(* IEC 61131-3 sources: inproshop/test13_exported/1.Function/FC, 5 files *)

(* ---- FC_AryCmp.st ---- *)
FUNCTION FC_AryCmp : BOOL
VAR_INPUT
	iAry1:ARRAY[0..50]OF BOOL;
	iAry2:ARRAY[0..50]OF BOOL;
END_VAR
VAR
	i: INT;
END_VAR

FOR i:=0 TO 50 BY 1 DO
	IF iAry1[i]<>iAry2[i] THEN
		FC_AryCmp:=FALSE;
		EXIT;
	END_IF;
	FC_AryCmp:=TRUE;
END_FOR

(* ---- FC_LCONCAT.st ---- *)
FUNCTION FC_LCONCAT : WSTRING//最终结果字符数量小于80
VAR_INPUT
	iSTR1:WSTRING;//输入1
	iSTR2:WSTRING;//输入2
END_VAR
VAR
	Num:INT;//用于循环变量
	Temp_Len:INT;//输入1字符串长度(偶数个)
	Temp_STR1:POINTER TO WSTRING;
	Temp_STR2:POINTER TO WSTRING;
	Temp_LCONCAT:POINTER TO WSTRING;

END_VAR

//wstring 变量合并
Temp_STR1:=ADR(iSTR1);//获取输入1地址
FOR Num:= 0 TO 80 BY 2 DO
	Temp_STR2:= Temp_STR1+INT_TO_DWORD(Num);
	IF Temp_STR2^="" THEN
		Temp_Len:=Num;//获取输入1长度
		EXIT;
	END_IF
END_FOR
Temp_LCONCAT:=ADR(FC_LCONCAT);
Temp_STR2:=Temp_LCONCAT+INT_TO_DWORD(Temp_Len);//获取输入2字符串存放开始地址
Temp_LCONCAT^:=iSTR1;//输入1字符串存放到对应地址
Temp_STR2^:=iSTR2;//输入2字符串存放到对应地址

(* ---- FC_StringSplit.st ---- *)
FUNCTION FC_StringSplit: BOOL
VAR_INPUT
	iSTR:STRING;//输入
	iCharSplit:STRING;//分割符
END_VAR
VAR_OUTPUT
	QSTR:ARRAY[0..10] OF STRING;//输出结果
END_VAR
VAR
	i:INT;//用于循环变量
	j:INT;//用于循环变量
	TotalCount:INT;
	tempIStr:STRING;
END_VAR

//string数据分解
j:=0;
TotalCount:=0;
TotalCount:=LEN(iSTR); //获取字符串长度
FOR i:=0 TO 10 BY 1 DO//字符串数组清空
	ClearString(QStr[i]);
END_FOR;
ClearString(tempIStr);
IF TotalCount<>0 THEN
		FOR i:=0 TO TotalCount   BY 1 DO
				tempIStr:=MID(iSTR,1,i);//提取字符
				IF tempIStr <> iCharSplit THEN  //分割条件
						QStr[j]:=CONCAT(QStr[j],tempIStr);//拼接字符
				ELSE
						j:=j+1;
				END_IF;
		END_FOR;
		FC_StringSplit:=TRUE;
ELSE
	FC_StringSplit:=FALSE;
END_IF;

(* ---- FC_SysTime.st ---- *)
FUNCTION FC_SysTime : BOOL
VAR_INPUT
	iNow:_sDT;
END_VAR
VAR_IN_OUT
	ioBefor:ARRAY[0..30]OF _sDT;
END_VAR
VAR
	i:UINT;
	uiMonth: INT;
END_VAR

ioBefor[0]:=iNow;
FOR i:=1 TO 30 BY 1 DO
	ioBefor[i]:=ioBefor[i-1];
	ioBefor[i].uiDay:=ioBefor[i-1].uiDay-1;

	IF ioBefor[i].uiDay=0 THEN
		CASE ioBefor[i-1].uiMonth OF
			1:
				ioBefor[i].uiDay:=31;
				ioBefor[i].uiMonth:=12;
				ioBefor[i].uiYear:=ioBefor[i-1].uiYear-1;
			2:
				ioBefor[i].uiDay:=31;
				ioBefor[i].uiMonth:=1;
			3:
				IF (ioBefor[i].uiYear MOD 4)=0 THEN
					ioBefor[i].uiDay:=29;
					ioBefor[i].uiMonth:=2;
				ELSE
					ioBefor[i].uiDay:=28;
					ioBefor[i].uiMonth:=2;
				END_IF
			4:
				ioBefor[i].uiDay:=31;
				ioBefor[i].uiMonth:=3;
			5:
				ioBefor[i].uiDay:=30;
				ioBefor[i].uiMonth:=4;
			6:
				ioBefor[i].uiDay:=31;
				ioBefor[i].uiMonth:=5;
			7:
				ioBefor[i].uiDay:=30;
				ioBefor[i].uiMonth:=6;

			8:
				ioBefor[i].uiDay:=31;
				ioBefor[i].uiMonth:=7;

			9:
				ioBefor[i].uiDay:=31;
				ioBefor[i].uiMonth:=8;

			10:
				ioBefor[i].uiDay:=30;
				ioBefor[i].uiMonth:=9;

			11:
				ioBefor[i].uiDay:=31;
				ioBefor[i].uiMonth:=10;

			12:
				ioBefor[i].uiDay:=30;
				ioBefor[i].uiMonth:=11;

		END_CASE

	END_IF
	ioBefor[i].uiDayOfWeek:=0;
	ioBefor[i].uiHour:=0;
	ioBefor[i].uiMinute:=0;
	ioBefor[i].uiSecond:=0;
	ioBefor[i].uiMillisecond:=0;
END_FOR

(* ---- FC_WStringSplit.st ---- *)
FUNCTION FC_WStringSplit:ARRAY[0..10] OF WSTRING
VAR_INPUT
	iwSTR:WSTRING;//输入1
	CharSplit:WSTRING;//分割符
END_VAR
VAR_OUTPUT
	QSTR1:ARRAY[0..10] OF WSTRING;//输出结果
END_VAR
VAR
	i:INT;//用于循环变量
	j:INT;//用于循环变量
	Temp_wSTR:ARRAY[0..100] OF Str_WstringWord;
END_VAR

//wstring 变量合并
j:=0;
FOR i:=0 TO 20 BY 1 DO
	QSTR1[i]:="";
END_FOR
FOR i:=0 TO 80 BY 1 DO
	Temp_wSTR[i].Wo:=iwSTR[i];
	IF Temp_wSTR[i].Ws<> "" THEN
		IF Temp_wSTR[i].Ws = CharSplit THEN
			j:=j+1;
		ELSE
			QSTR1[j]:=FC_LCONCAT(QSTR1[j],Temp_wSTR[i].Ws);
		END_IF
		;
	ELSE
		EXIT;
	END_IF
END_FOR
